FUNCTION_BLOCK FB_SequenceGET_READY_EXTEND EXTENDS FB_SequenceBase



VAR_IN_OUT
	devices: ST_POPComponents;
END_VAR

METHOD FB_init : BOOL
VAR_INPUT
	bInitRetains : BOOL; // if TRUE, the retain variables are initialized (warm start / cold start)
	bInCopyCode : BOOL;  // if TRUE, the instance afterwards gets moved into the copy code (online change)
	
	
END_VAR
(*
		Here we set the order of things to command, what the commands should be, and also how much time to allow during and between steps
		Every component listed below becomes 'Enabled' at each step
*)
sSequenceName:= 'POP Conveyor Reverse Sequence';
sSequenceDescription := 'Performs the full reverse series of actions (starting with lifting movement and followed by static conveyors';
bSequentional_1_Flood_0 := TRUE;
END_METHOD

METHOD populateSteps : ST_SequenceStep
VAR_INPUT
	
END_VAR
(*
		Here we set the order of things to command, what the commands should be, and also how much time to allow during and between steps
		Every component listed below becomes 'Enabled' at each step
*)

Step1.Device := devices.fbLinAct_POP1;
Step1.Command := E_DeviceState.EXTENDED;
Step1.StepMinDuration := T#0S; 
Step1.DelayUntilNextStep := T#0S;
Step1.WaitForAction := FALSE;
aSequenceSteps[1] :=   Step1;

Step2.Device := devices.fbLinAct_POP1;
Step2.Command := E_DeviceState.EXTENDED;
Step2.StepMinDuration := T#0S; 
Step2.DelayUntilNextStep := T#0S;
Step2.WaitForAction := FALSE;
aSequenceSteps[2] :=   Step2;

Step3.Device := devices.fbLinAct_POP2;
Step3.Command := E_DeviceState.EXTENDED;
Step3.StepMinDuration := T#0S;
Step3.DelayUntilNextStep := T#0S;
Step3.WaitForAction := FALSE;
aSequenceSteps[3] :=   Step3;

Step4.Device := devices.fbTrayCentre_POP1;
Step4.Command := E_DeviceState.RETRACTED;
Step4.StepMinDuration := T#0S;
Step4.DelayUntilNextStep := T#0S;
Step4.WaitForAction := FALSE;
aSequenceSteps[4] :=   Step4;

Step5.Device := devices.fbTrayCentre_POP2;
Step5.Command := E_DeviceState.RETRACTED;
Step5.StepMinDuration := T#0S;
Step5.DelayUntilNextStep := T#0S;
Step5.WaitForAction := FALSE;
aSequenceSteps[5] :=   Step5;

Step6.Device := devices.fbTrayCentre_POP3;
Step6.Command := E_DeviceState.RETRACTED;
Step6.StepMinDuration := T#0S;
Step6.DelayUntilNextStep := T#0S;
Step6.WaitForAction := FALSE;
aSequenceSteps[6] :=   Step6;

nNumberSequenceSteps := 6;  // use this number to limit the number of operations
updateVarIDs();
END_METHOD

END_FUNCTION_BLOCK

(* stored: Version 1.1.0.1, ProductVersion 3.1.4024.12
   POU FB_SequenceGET_READY_EXTEND: Id {952f6079-71bd-4c41-9ff1-8837d563b3de}, SpecialFunc None
   Method FB_init: Id {c4d2c01d-4d77-44d5-9ad4-3d6eb60085e0}
   Method populateSteps: Id {0c905f04-472a-4f64-8146-9e1a0a1c577a} *)
